{attribute addProperty BoxType "EL6201-0000-0017"}
{attribute addProperty Id "Slave_11A_DO0BIT10.12581Slave_11A_DO1BIT10.12582Slave_11A_DO2BIT10.12583Slave_11A_DO3BIT10.12584Slave_11B_DO0BIT10.12585Slave_11B_DO1BIT10.12586Slave_11B_DO2BIT10.12587Slave_11B_DO3BIT10.12588"}
{attribute addProperty CRC "574970854"}
{attribute addProperty SizeInBites "8"}
{attribute addProperty SizeInBytes "1"}
TYPE Slave_11_Outputs_22455BE6 :
STRUCT
	{attribute addProperty Name "Slave_11A_DO0"}
	Slave_11A_DO0 : BIT;
	{attribute addProperty Name "Slave_11A_DO1"}
	Slave_11A_DO1 : BIT;
	{attribute addProperty Name "Slave_11A_DO2"}
	Slave_11A_DO2 : BIT;
	{attribute addProperty Name "Slave_11A_DO3"}
	Slave_11A_DO3 : BIT;
	{attribute addProperty Name "Slave_11B_DO0"}
	Slave_11B_DO0 : BIT;
	{attribute addProperty Name "Slave_11B_DO1"}
	Slave_11B_DO1 : BIT;
	{attribute addProperty Name "Slave_11B_DO2"}
	Slave_11B_DO2 : BIT;
	{attribute addProperty Name "Slave_11B_DO3"}
	Slave_11B_DO3 : BIT;
END_STRUCT
END_TYPE

(* stored: Version 1.2.0.0, ProductVersion 3.1.4024.9
   DUT Slave_11_Outputs_22455BE6: Id {7573b0ff-32f9-420a-b8e7-92accc5c5b03} *)
